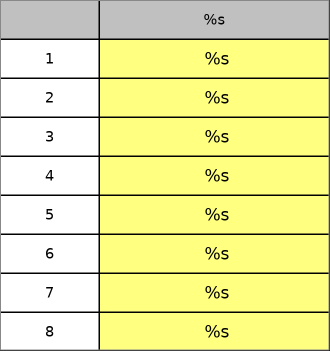
VISUALIZATION VISU_CONF_BAL  // 330x351
VAR_IN_OUT
	m_Input_SWEEP : BLOCK_TELEMARK_CHEETAH_SWEEP;
END_VAR
    Rectangle (0,0 99x39)
    Rectangle (99,39 231x39), "%s", text variable: m_Input_SWEEP.PRM_BAL[1], input disabled if: NOT Global_Variables.PRG_USER.ACTU_USER.CONF_MACHINE
        OnMouseDown: write the text variable via InputWithLimits
    Rectangle (99,0 231x39), "%s", text list: 'TextList_Config_Evap', text index: 8
    Rectangle (0,39 99x39), "1"
    Rectangle (0,78 99x39), "2"
    Rectangle (99,78 231x39), "%s", text variable: m_Input_SWEEP.PRM_BAL[2], input disabled if: NOT Global_Variables.PRG_USER.ACTU_USER.CONF_MACHINE
        OnMouseDown: write the text variable via InputWithLimits
    Rectangle (0,117 99x39), "3"
    Rectangle (99,117 231x39), "%s", text variable: m_Input_SWEEP.PRM_BAL[3], input disabled if: NOT Global_Variables.PRG_USER.ACTU_USER.CONF_MACHINE
        OnMouseDown: write the text variable via InputWithLimits
    Rectangle (0,156 99x39), "4"
    Rectangle (99,156 231x39), "%s", text variable: m_Input_SWEEP.PRM_BAL[4], input disabled if: NOT Global_Variables.PRG_USER.ACTU_USER.CONF_MACHINE
        OnMouseDown: write the text variable via InputWithLimits
    Rectangle (99,195 231x39), "%s", text variable: m_Input_SWEEP.PRM_BAL[5], input disabled if: NOT Global_Variables.PRG_USER.ACTU_USER.CONF_MACHINE
        OnMouseDown: write the text variable via InputWithLimits
    Rectangle (0,195 99x39), "5"
    Rectangle (0,234 99x39), "6"
    Rectangle (99,234 231x39), "%s", text variable: m_Input_SWEEP.PRM_BAL[6], input disabled if: NOT Global_Variables.PRG_USER.ACTU_USER.CONF_MACHINE
        OnMouseDown: write the text variable via InputWithLimits
    Rectangle (0,273 99x39), "7"
    Rectangle (99,273 231x39), "%s", text variable: m_Input_SWEEP.PRM_BAL[7], input disabled if: NOT Global_Variables.PRG_USER.ACTU_USER.CONF_MACHINE
        OnMouseDown: write the text variable via InputWithLimits
    Rectangle (0,312 99x39), "8"
    Rectangle (99,312 231x39), "%s", text variable: m_Input_SWEEP.PRM_BAL[8], input disabled if: NOT Global_Variables.PRG_USER.ACTU_USER.CONF_MACHINE
        OnMouseDown: write the text variable via InputWithLimits
END_VISUALIZATION

(* stored: Version 1.1.0.1, ProductVersion 3.1.4026.18
   Visu VISU_CONF_BAL: Id {f07d901d-424a-4de7-a820-1190fc017a87} *)
